// TIA Portal V20 export
DATA_BLOCK "idbConveyor"   // DB2
// stored: InstanceOfName Conveyor4.Conveyor_C4, InstanceOfType FB, Namespace Conveyor4
"Conveyor4.Conveyor_C4"
   // VAR
   //    statManRight : Bool;
   //    statManLeft : Bool;
   //    statAutoRight : Bool;
   //    statAutoLeft : Bool;
   //    statRunning : Bool;
   //    reLightBarrier { S7_SetPoint := 'True'} : R_TRIG;
   //    tonDelayStart { S7_SetPoint := 'True'} : TON_TIME;
   // END_VAR
BEGIN
END_DATA_BLOCK
